// TIA Portal V20 export
ORGANIZATION_BLOCK "Startup"   // OB1060, LAD, Startup
TITLE = "Complete Restart"
AUTHOR : ERsystem_FA2_DH. Kim
// stored: AutoNumber false, IsIECCheckEnabled true, Namespace Unit1.Em6, SetENOAutomatically false
   VAR_INPUT
      LostRetentive : Bool;   // True if retentive data are lost
      LostRTC : Bool;   // True if date and time are lost
   END_VAR
BEGIN

REGION Network 1 (SCL): Build the Absolut Reference Designator
   // Set the Absoult Reference Designator in the Config DB
   IF LEN(IN := "Unit1.Em6.Config".em.referenceDesignator.parent) <> 0 THEN
     "Unit1.Em6.Config".em.referenceDesignator.combined := CONCAT_WSTRING(IN1 := "Unit1.Em6.Config".em.referenceDesignator.parent, IN2 := WSTRING#'.', IN3 := "Unit1.Em6.Config".em.referenceDesignator.relative);
   ELSE
     "Unit1.Em6.Config".em.referenceDesignator.combined := "Unit1.Em6.Config".em.referenceDesignator.relative;
   END_IF;
END_REGION

REGION Network 2 (SCL): Assign axes data
   //Assign axes
   "Unit1.Em6.Config".axis[1] := "BA030AZSCDR21_FinalRollerFrontAxisX";
   "Unit1.Em6.Config".axis[2] := "BA030AZSCDR22_FinalRollerRearAxisX";
   "Unit1.Em6.Config".axis[3] := "BA030AZSCDR23_MendrelAnodeFrontAxisY";
   "Unit1.Em6.Config".axis[4] := "BA030AZSCDR24_MendrelAnodeFrontAxisZ";
   "Unit1.Em6.Config".axis[5] := "BA030AZSCDR25_MendrelAnodeRearAxisY";
   "Unit1.Em6.Config".axis[6] := "BA030AZSCDR26_MendrelAnodeRearAxisZ";
   "Unit1.Em6.Config".axis[7] := "BA030AZSCDR27_MendrelCathodeFrontAxisY";
   "Unit1.Em6.Config".axis[8] := "BA030AZSCDR28_MendrelCathodeFrontAxisZ";
   "Unit1.Em6.Config".axis[9] := "BA030AZSCDR29_MendrelCathodeRearAxisY";
   "Unit1.Em6.Config".axis[10] := "BA030AZSCDR30_MendrelCathodeRearAxisZ";
   "Unit1.Em6.Config".axis[11] := "BA030AZSCDR31_StackTableAxisZ";
   "Unit1.Em6.Config".axis[12] := "BA030AZSCDR32_StackTableOutFrontAxisZ";
   "Unit1.Em6.Config".axis[13] := "BA030AZSCDR33_StackTableOutRearAxisZ";
   "Unit1.Em6.Config".axis[14] := "BA030A_MasterAxis";

   // Config.cam[1] := _.BA030AZSCDR21_FinalRollerFrontXCamMain;
   // Config.cam[2] := _.BA030AZSCDR23_MendrelAnodeFrontAxisYCamMain;
   // Config.cam[3] := _.BA030AZSCDR24_MendrelAnodeFrontAxisZCamMain;
   // Config.cam[4] := _.BA030AZSCDR25_MendrelAnodeRearAxisYCamMain;
   // Config.cam[5] := _.BA030AZSCDR26_MendrelAnodeRearAxisZCamMain;
   // Config.cam[6] := _.BA030AZSCDR23_MendrelCathodeFrontAxisYCamMain;
   // Config.cam[7] := _.BA030AZSCDR24_MendrelCathodeFrontAxisZCamMain;
   // Config.cam[8] := _.BA030AZSCDR25_MendrelCathodeRearAxisYCamMain;
   // Config.cam[9] := _.BA030AZSCDR26_MendrelCathodeRearAxisZCamMain;

   // FB Enable
   "Unit1.Em6.HmiInterface".cmFinalRollerFrontAxisX.commands.enableMasterControl := TRUE;
   "Unit1.Em6.HmiInterface".cmFinalRollerRearAxisX.commands.enableMasterControl := TRUE;
   "Unit1.Em6.HmiInterface".cmMendrelAnodeFrontAxisY.commands.enableMasterControl := TRUE;
   "Unit1.Em6.HmiInterface".cmMendrelAnodeFrontAxisZ.commands.enableMasterControl := TRUE;
   "Unit1.Em6.HmiInterface".cmMendrelAnodeRearAxisY.commands.enableMasterControl := TRUE;
   "Unit1.Em6.HmiInterface".cmMendrelAnodeRearAxisZ.commands.enableMasterControl := TRUE;
   "Unit1.Em6.HmiInterface".cmMendrelCathodeFrontAxisY.commands.enableMasterControl := TRUE;
   "Unit1.Em6.HmiInterface".cmMendrelCathodeFrontAxisZ.commands.enableMasterControl := TRUE;
   "Unit1.Em6.HmiInterface".cmMendrelCathodeRearAxisY.commands.enableMasterControl := TRUE;
   "Unit1.Em6.HmiInterface".cmMendrelCathodeRearAxisZ.commands.enableMasterControl := TRUE;
   "Unit1.Em6.HmiInterface".cmStackTableAxisZ.commands.enableMasterControl := TRUE;
   "Unit1.Em6.HmiInterface".cmStackTableOutFrontAxisZ.commands.enableMasterControl := TRUE;
   "Unit1.Em6.HmiInterface".cmStackTableOutRearAxisZ.commands.enableMasterControl := TRUE;

   // Axis 1 BA040AZSCDR21_FinalRollerFrontAxisX
   "Unit1.Em6.HmiInterface".cmFinalRollerFrontAxisX.commandConfiguration.jog.velocity := 10.0;
   "Unit1.Em6.HmiInterface".cmFinalRollerFrontAxisX.commandConfiguration.jog.acceleration := 100.0;
   "Unit1.Em6.HmiInterface".cmFinalRollerFrontAxisX.commandConfiguration.jog.deceleration := 100.0;
   "Unit1.Em6.HmiInterface".cmFinalRollerFrontAxisX.commandConfiguration.moveVelocity.velocity := 10.0;
   "Unit1.Em6.HmiInterface".cmFinalRollerFrontAxisX.commandConfiguration.moveVelocity.acceleration := 100.0;
   "Unit1.Em6.HmiInterface".cmFinalRollerFrontAxisX.commandConfiguration.moveVelocity.deceleration := 100.0;
   "Unit1.Em6.HmiInterface".cmFinalRollerFrontAxisX.commandConfiguration.posRelative.velocity := 10.0;
   "Unit1.Em6.HmiInterface".cmFinalRollerFrontAxisX.commandConfiguration.posRelative.acceleration := 100.0;
   "Unit1.Em6.HmiInterface".cmFinalRollerFrontAxisX.commandConfiguration.posRelative.deceleration := 100.0;
   "Unit1.Em6.HmiInterface".cmFinalRollerFrontAxisX.configuration.setPositions[0].name := 'cathode';
   "Unit1.Em6.HmiInterface".cmFinalRollerFrontAxisX.configuration.setPositions[1].name := 'anode';

   // Axis 2 BA040AZSCDR22_FinalRollerRearAxisX
   "Unit1.Em6.HmiInterface".cmFinalRollerRearAxisX.commandConfiguration.jog.velocity := 10.0;
   "Unit1.Em6.HmiInterface".cmFinalRollerRearAxisX.commandConfiguration.jog.acceleration := 100.0;
   "Unit1.Em6.HmiInterface".cmFinalRollerRearAxisX.commandConfiguration.jog.deceleration := 100.0;
   "Unit1.Em6.HmiInterface".cmFinalRollerRearAxisX.commandConfiguration.moveVelocity.velocity := 10.0;
   "Unit1.Em6.HmiInterface".cmFinalRollerRearAxisX.commandConfiguration.moveVelocity.acceleration := 100.0;
   "Unit1.Em6.HmiInterface".cmFinalRollerRearAxisX.commandConfiguration.moveVelocity.deceleration := 100.0;
   "Unit1.Em6.HmiInterface".cmFinalRollerRearAxisX.commandConfiguration.posRelative.velocity := 10.0;
   "Unit1.Em6.HmiInterface".cmFinalRollerRearAxisX.commandConfiguration.posRelative.acceleration := 100.0;
   "Unit1.Em6.HmiInterface".cmFinalRollerRearAxisX.commandConfiguration.posRelative.deceleration := 100.0;
   "Unit1.Em6.HmiInterface".cmFinalRollerRearAxisX.configuration.setPositions[0].name := 'cathode';
   "Unit1.Em6.HmiInterface".cmFinalRollerRearAxisX.configuration.setPositions[1].name := 'anode';

   // Axis 3 BA040AZSCDR23_MendrelAnodeFrontAxisY
   "Unit1.Em6.HmiInterface".cmMendrelAnodeFrontAxisY.commandConfiguration.jog.velocity := 10.0;
   "Unit1.Em6.HmiInterface".cmMendrelAnodeFrontAxisY.commandConfiguration.jog.acceleration := 100.0;
   "Unit1.Em6.HmiInterface".cmMendrelAnodeFrontAxisY.commandConfiguration.jog.deceleration := 100.0;
   "Unit1.Em6.HmiInterface".cmMendrelAnodeFrontAxisY.commandConfiguration.moveVelocity.velocity := 10.0;
   "Unit1.Em6.HmiInterface".cmMendrelAnodeFrontAxisY.commandConfiguration.moveVelocity.acceleration := 100.0;
   "Unit1.Em6.HmiInterface".cmMendrelAnodeFrontAxisY.commandConfiguration.moveVelocity.deceleration := 100.0;
   "Unit1.Em6.HmiInterface".cmMendrelAnodeFrontAxisY.commandConfiguration.posRelative.velocity := 10.0;
   "Unit1.Em6.HmiInterface".cmMendrelAnodeFrontAxisY.commandConfiguration.posRelative.acceleration := 100.0;
   "Unit1.Em6.HmiInterface".cmMendrelAnodeFrontAxisY.commandConfiguration.posRelative.deceleration := 100.0;
   "Unit1.Em6.HmiInterface".cmMendrelAnodeFrontAxisY.configuration.setPositions[0].name := 'backward';
   "Unit1.Em6.HmiInterface".cmMendrelAnodeFrontAxisY.configuration.setPositions[1].name := 'forward';

   // Axis 4 BA040AZSCDR24_MendrelAnodeFrontAxisZ
   "Unit1.Em6.HmiInterface".cmMendrelAnodeFrontAxisZ.commandConfiguration.jog.velocity := 10.0;
   "Unit1.Em6.HmiInterface".cmMendrelAnodeFrontAxisZ.commandConfiguration.jog.acceleration := 100.0;
   "Unit1.Em6.HmiInterface".cmMendrelAnodeFrontAxisZ.commandConfiguration.jog.deceleration := 100.0;
   "Unit1.Em6.HmiInterface".cmMendrelAnodeFrontAxisZ.commandConfiguration.moveVelocity.velocity := 10.0;
   "Unit1.Em6.HmiInterface".cmMendrelAnodeFrontAxisZ.commandConfiguration.moveVelocity.acceleration := 100.0;
   "Unit1.Em6.HmiInterface".cmMendrelAnodeFrontAxisZ.commandConfiguration.moveVelocity.deceleration := 100.0;
   "Unit1.Em6.HmiInterface".cmMendrelAnodeFrontAxisZ.commandConfiguration.posRelative.velocity := 10.0;
   "Unit1.Em6.HmiInterface".cmMendrelAnodeFrontAxisZ.commandConfiguration.posRelative.acceleration := 100.0;
   "Unit1.Em6.HmiInterface".cmMendrelAnodeFrontAxisZ.commandConfiguration.posRelative.deceleration := 100.0;
   "Unit1.Em6.HmiInterface".cmMendrelAnodeFrontAxisZ.configuration.setPositions[0].name := 'up';
   "Unit1.Em6.HmiInterface".cmMendrelAnodeFrontAxisZ.configuration.setPositions[1].name := 'down';

   // Axis 5 BA040AZSCDR25_MendrelAnodeRearAxisY
   "Unit1.Em6.HmiInterface".cmMendrelAnodeRearAxisY.commandConfiguration.jog.velocity := 10.0;
   "Unit1.Em6.HmiInterface".cmMendrelAnodeRearAxisY.commandConfiguration.jog.acceleration := 100.0;
   "Unit1.Em6.HmiInterface".cmMendrelAnodeRearAxisY.commandConfiguration.jog.deceleration := 100.0;
   "Unit1.Em6.HmiInterface".cmMendrelAnodeRearAxisY.commandConfiguration.moveVelocity.velocity := 10.0;
   "Unit1.Em6.HmiInterface".cmMendrelAnodeRearAxisY.commandConfiguration.moveVelocity.acceleration := 100.0;
   "Unit1.Em6.HmiInterface".cmMendrelAnodeRearAxisY.commandConfiguration.moveVelocity.deceleration := 100.0;
   "Unit1.Em6.HmiInterface".cmMendrelAnodeRearAxisY.commandConfiguration.posRelative.velocity := 10.0;
   "Unit1.Em6.HmiInterface".cmMendrelAnodeRearAxisY.commandConfiguration.posRelative.acceleration := 100.0;
   "Unit1.Em6.HmiInterface".cmMendrelAnodeRearAxisY.commandConfiguration.posRelative.deceleration := 100.0;
   "Unit1.Em6.HmiInterface".cmMendrelAnodeRearAxisY.configuration.setPositions[0].name := 'backward';
   "Unit1.Em6.HmiInterface".cmMendrelAnodeRearAxisY.configuration.setPositions[1].name := 'forward';

   // Axis 6 BA040AZSCDR26_MendrelAnodeRearAxisZ
   "Unit1.Em6.HmiInterface".cmMendrelAnodeRearAxisZ.commandConfiguration.jog.velocity := 10.0;
   "Unit1.Em6.HmiInterface".cmMendrelAnodeRearAxisZ.commandConfiguration.jog.acceleration := 100.0;
   "Unit1.Em6.HmiInterface".cmMendrelAnodeRearAxisZ.commandConfiguration.jog.deceleration := 100.0;
   "Unit1.Em6.HmiInterface".cmMendrelAnodeRearAxisZ.commandConfiguration.moveVelocity.velocity := 10.0;
   "Unit1.Em6.HmiInterface".cmMendrelAnodeRearAxisZ.commandConfiguration.moveVelocity.acceleration := 100.0;
   "Unit1.Em6.HmiInterface".cmMendrelAnodeRearAxisZ.commandConfiguration.moveVelocity.deceleration := 100.0;
   "Unit1.Em6.HmiInterface".cmMendrelAnodeRearAxisZ.commandConfiguration.posRelative.velocity := 10.0;
   "Unit1.Em6.HmiInterface".cmMendrelAnodeRearAxisZ.commandConfiguration.posRelative.acceleration := 100.0;
   "Unit1.Em6.HmiInterface".cmMendrelAnodeRearAxisZ.commandConfiguration.posRelative.deceleration := 100.0;
   "Unit1.Em6.HmiInterface".cmMendrelAnodeRearAxisZ.configuration.setPositions[0].name := 'up';
   "Unit1.Em6.HmiInterface".cmMendrelAnodeRearAxisZ.configuration.setPositions[1].name := 'down';

   // Axis 7 BA040AZSCDR27_MendrelCathodeFrontAxisY
   "Unit1.Em6.HmiInterface".cmMendrelCathodeFrontAxisY.commandConfiguration.jog.velocity := 10.0;
   "Unit1.Em6.HmiInterface".cmMendrelCathodeFrontAxisY.commandConfiguration.jog.acceleration := 100.0;
   "Unit1.Em6.HmiInterface".cmMendrelCathodeFrontAxisY.commandConfiguration.jog.deceleration := 100.0;
   "Unit1.Em6.HmiInterface".cmMendrelCathodeFrontAxisY.commandConfiguration.moveVelocity.velocity := 10.0;
   "Unit1.Em6.HmiInterface".cmMendrelCathodeFrontAxisY.commandConfiguration.moveVelocity.acceleration := 100.0;
   "Unit1.Em6.HmiInterface".cmMendrelCathodeFrontAxisY.commandConfiguration.moveVelocity.deceleration := 100.0;
   "Unit1.Em6.HmiInterface".cmMendrelCathodeFrontAxisY.commandConfiguration.posRelative.velocity := 10.0;
   "Unit1.Em6.HmiInterface".cmMendrelCathodeFrontAxisY.commandConfiguration.posRelative.acceleration := 100.0;
   "Unit1.Em6.HmiInterface".cmMendrelCathodeFrontAxisY.commandConfiguration.posRelative.deceleration := 100.0;
   "Unit1.Em6.HmiInterface".cmMendrelCathodeFrontAxisY.configuration.setPositions[0].name := 'backward';
   "Unit1.Em6.HmiInterface".cmMendrelCathodeFrontAxisY.configuration.setPositions[1].name := 'forward';

   // Axis 8 BA040AZSCDR28_MendrelCathodeFrontAxisZ
   "Unit1.Em6.HmiInterface".cmMendrelCathodeFrontAxisZ.commandConfiguration.jog.velocity := 10.0;
   "Unit1.Em6.HmiInterface".cmMendrelCathodeFrontAxisZ.commandConfiguration.jog.acceleration := 100.0;
   "Unit1.Em6.HmiInterface".cmMendrelCathodeFrontAxisZ.commandConfiguration.jog.deceleration := 100.0;
   "Unit1.Em6.HmiInterface".cmMendrelCathodeFrontAxisZ.commandConfiguration.moveVelocity.velocity := 10.0;
   "Unit1.Em6.HmiInterface".cmMendrelCathodeFrontAxisZ.commandConfiguration.moveVelocity.acceleration := 100.0;
   "Unit1.Em6.HmiInterface".cmMendrelCathodeFrontAxisZ.commandConfiguration.moveVelocity.deceleration := 100.0;
   "Unit1.Em6.HmiInterface".cmMendrelCathodeFrontAxisZ.commandConfiguration.posRelative.velocity := 10.0;
   "Unit1.Em6.HmiInterface".cmMendrelCathodeFrontAxisZ.commandConfiguration.posRelative.acceleration := 100.0;
   "Unit1.Em6.HmiInterface".cmMendrelCathodeFrontAxisZ.commandConfiguration.posRelative.deceleration := 100.0;
   "Unit1.Em6.HmiInterface".cmMendrelCathodeFrontAxisZ.configuration.setPositions[0].name := 'up';
   "Unit1.Em6.HmiInterface".cmMendrelCathodeFrontAxisZ.configuration.setPositions[1].name := 'down';

   // Axis 9 BA040AZSCDR29_MendrelCathodeRearAxisY
   "Unit1.Em6.HmiInterface".cmMendrelCathodeRearAxisY.commandConfiguration.jog.velocity := 10.0;
   "Unit1.Em6.HmiInterface".cmMendrelCathodeRearAxisY.commandConfiguration.jog.acceleration := 100.0;
   "Unit1.Em6.HmiInterface".cmMendrelCathodeRearAxisY.commandConfiguration.jog.deceleration := 100.0;
   "Unit1.Em6.HmiInterface".cmMendrelCathodeRearAxisY.commandConfiguration.moveVelocity.velocity := 10.0;
   "Unit1.Em6.HmiInterface".cmMendrelCathodeRearAxisY.commandConfiguration.moveVelocity.acceleration := 100.0;
   "Unit1.Em6.HmiInterface".cmMendrelCathodeRearAxisY.commandConfiguration.moveVelocity.deceleration := 100.0;
   "Unit1.Em6.HmiInterface".cmMendrelCathodeRearAxisY.commandConfiguration.posRelative.velocity := 10.0;
   "Unit1.Em6.HmiInterface".cmMendrelCathodeRearAxisY.commandConfiguration.posRelative.acceleration := 100.0;
   "Unit1.Em6.HmiInterface".cmMendrelCathodeRearAxisY.commandConfiguration.posRelative.deceleration := 100.0;
   "Unit1.Em6.HmiInterface".cmMendrelCathodeRearAxisY.configuration.setPositions[0].name := 'backward';
   "Unit1.Em6.HmiInterface".cmMendrelCathodeRearAxisY.configuration.setPositions[1].name := 'forward';

   // Axis 10 BA040AZSCDR30_MendrelCathodeRearAxisZ
   "Unit1.Em6.HmiInterface".cmMendrelCathodeRearAxisZ.commandConfiguration.jog.velocity := 10.0;
   "Unit1.Em6.HmiInterface".cmMendrelCathodeRearAxisZ.commandConfiguration.jog.acceleration := 100.0;
   "Unit1.Em6.HmiInterface".cmMendrelCathodeRearAxisZ.commandConfiguration.jog.deceleration := 100.0;
   "Unit1.Em6.HmiInterface".cmMendrelCathodeRearAxisZ.commandConfiguration.moveVelocity.velocity := 10.0;
   "Unit1.Em6.HmiInterface".cmMendrelCathodeRearAxisZ.commandConfiguration.moveVelocity.acceleration := 100.0;
   "Unit1.Em6.HmiInterface".cmMendrelCathodeRearAxisZ.commandConfiguration.moveVelocity.deceleration := 100.0;
   "Unit1.Em6.HmiInterface".cmMendrelCathodeRearAxisZ.commandConfiguration.posRelative.velocity := 10.0;
   "Unit1.Em6.HmiInterface".cmMendrelCathodeRearAxisZ.commandConfiguration.posRelative.acceleration := 100.0;
   "Unit1.Em6.HmiInterface".cmMendrelCathodeRearAxisZ.commandConfiguration.posRelative.deceleration := 100.0;
   "Unit1.Em6.HmiInterface".cmMendrelCathodeRearAxisZ.configuration.setPositions[0].name := 'up';
   "Unit1.Em6.HmiInterface".cmMendrelCathodeRearAxisZ.configuration.setPositions[1].name := 'down';

   // Axis 11 BA040AZSCDR31_StackTableAxisZ
   "Unit1.Em6.HmiInterface".cmStackTableAxisZ.commandConfiguration.jog.velocity := 10.0;
   "Unit1.Em6.HmiInterface".cmStackTableAxisZ.commandConfiguration.jog.acceleration := 100.0;
   "Unit1.Em6.HmiInterface".cmStackTableAxisZ.commandConfiguration.jog.deceleration := 100.0;
   "Unit1.Em6.HmiInterface".cmStackTableAxisZ.commandConfiguration.moveVelocity.velocity := 10.0;
   "Unit1.Em6.HmiInterface".cmStackTableAxisZ.commandConfiguration.moveVelocity.acceleration := 100.0;
   "Unit1.Em6.HmiInterface".cmStackTableAxisZ.commandConfiguration.moveVelocity.deceleration := 100.0;
   "Unit1.Em6.HmiInterface".cmStackTableAxisZ.commandConfiguration.posRelative.velocity := 10.0;
   "Unit1.Em6.HmiInterface".cmStackTableAxisZ.commandConfiguration.posRelative.acceleration := 100.0;
   "Unit1.Em6.HmiInterface".cmStackTableAxisZ.commandConfiguration.posRelative.deceleration := 100.0;
   "Unit1.Em6.HmiInterface".cmStackTableAxisZ.configuration.setPositions[0].name := 'wait';
   "Unit1.Em6.HmiInterface".cmStackTableAxisZ.configuration.setPositions[1].name := 'currentJRThickness';
   "Unit1.Em6.HmiInterface".cmStackTableAxisZ.configuration.setPositions[2].name := 'fullJRThickness';

   // Axis 12 BA040AZSCDR32_StackTableOutFrontAxisZ
   "Unit1.Em6.HmiInterface".cmStackTableOutFrontAxisZ.commandConfiguration.jog.velocity := 10.0;
   "Unit1.Em6.HmiInterface".cmStackTableOutFrontAxisZ.commandConfiguration.jog.acceleration := 100.0;
   "Unit1.Em6.HmiInterface".cmStackTableOutFrontAxisZ.commandConfiguration.jog.deceleration := 100.0;
   "Unit1.Em6.HmiInterface".cmStackTableOutFrontAxisZ.commandConfiguration.moveVelocity.velocity := 10.0;
   "Unit1.Em6.HmiInterface".cmStackTableOutFrontAxisZ.commandConfiguration.moveVelocity.acceleration := 100.0;
   "Unit1.Em6.HmiInterface".cmStackTableOutFrontAxisZ.commandConfiguration.moveVelocity.deceleration := 100.0;
   "Unit1.Em6.HmiInterface".cmStackTableOutFrontAxisZ.commandConfiguration.posRelative.velocity := 10.0;
   "Unit1.Em6.HmiInterface".cmStackTableOutFrontAxisZ.commandConfiguration.posRelative.acceleration := 100.0;
   "Unit1.Em6.HmiInterface".cmStackTableOutFrontAxisZ.commandConfiguration.posRelative.deceleration := 100.0;
   "Unit1.Em6.HmiInterface".cmStackTableOutFrontAxisZ.configuration.setPositions[0].name := 'down';
   "Unit1.Em6.HmiInterface".cmStackTableOutFrontAxisZ.configuration.setPositions[1].name := 'up';

   // Axis 13 BA040AZSCDR33_StackTableOutRearAxisZ
   "Unit1.Em6.HmiInterface".cmStackTableOutRearAxisZ.commandConfiguration.jog.velocity := 10.0;
   "Unit1.Em6.HmiInterface".cmStackTableOutRearAxisZ.commandConfiguration.jog.acceleration := 100.0;
   "Unit1.Em6.HmiInterface".cmStackTableOutRearAxisZ.commandConfiguration.jog.deceleration := 100.0;
   "Unit1.Em6.HmiInterface".cmStackTableOutRearAxisZ.commandConfiguration.moveVelocity.velocity := 10.0;
   "Unit1.Em6.HmiInterface".cmStackTableOutRearAxisZ.commandConfiguration.moveVelocity.acceleration := 100.0;
   "Unit1.Em6.HmiInterface".cmStackTableOutRearAxisZ.commandConfiguration.moveVelocity.deceleration := 100.0;
   "Unit1.Em6.HmiInterface".cmStackTableOutRearAxisZ.commandConfiguration.posRelative.velocity := 10.0;
   "Unit1.Em6.HmiInterface".cmStackTableOutRearAxisZ.commandConfiguration.posRelative.acceleration := 100.0;
   "Unit1.Em6.HmiInterface".cmStackTableOutRearAxisZ.commandConfiguration.posRelative.deceleration := 100.0;
   "Unit1.Em6.HmiInterface".cmStackTableOutRearAxisZ.configuration.setPositions[0].name := 'down';
   "Unit1.Em6.HmiInterface".cmStackTableOutRearAxisZ.configuration.setPositions[1].name := 'up';
END_REGION

REGION Network 3 (SCL): Assign TwoWayActuator data
   //Assign Configuration data of TwoWayActuator

   //cmMendrelAnodeFrontClamp
   "Unit1.Em6.Config".cmMendrelAnodeFrontClamp.referenceDesignator := WSTRING#'AnodeFrontClamp';
   "Unit1.Em6.Config".cmMendrelAnodeFrontClamp.disableFeedbackHomePos := TRUE;
   "Unit1.Em6.Config".cmMendrelAnodeFrontClamp.disableFeedbackWorkPos := TRUE;
   "Unit1.Em6.HmiInterface".cmMendrelAnodeFrontClamp.configuration.referenceDesignator := WSTRING#'AnodeFrontClamp';
   "Unit1.Em6.HmiInterface".cmMendrelAnodeFrontClamp.configuration.disableFeedbackHomePos := TRUE;
   "Unit1.Em6.HmiInterface".cmMendrelAnodeFrontClamp.configuration.disableFeedbackWorkPos := TRUE;

   //cmMendrelAnodeRearClamp
   "Unit1.Em6.Config".cmMendrelAnodeRearClamp.referenceDesignator := WSTRING#'AnodeRearClamp';
   "Unit1.Em6.Config".cmMendrelAnodeRearClamp.disableFeedbackHomePos := TRUE;
   "Unit1.Em6.Config".cmMendrelAnodeRearClamp.disableFeedbackWorkPos := TRUE;
   "Unit1.Em6.HmiInterface".cmMendrelAnodeRearClamp.configuration.referenceDesignator := WSTRING#'AnodeRearClamp';
   "Unit1.Em6.HmiInterface".cmMendrelAnodeRearClamp.configuration.disableFeedbackHomePos := TRUE;
   "Unit1.Em6.HmiInterface".cmMendrelAnodeRearClamp.configuration.disableFeedbackWorkPos := TRUE;

   //cmMendrelCathodeFrontClamp
   "Unit1.Em6.Config".cmMendrelCathodeFrontClamp.referenceDesignator := WSTRING#'CathodeFrontClamp';
   "Unit1.Em6.Config".cmMendrelCathodeFrontClamp.disableFeedbackHomePos := TRUE;
   "Unit1.Em6.Config".cmMendrelCathodeFrontClamp.disableFeedbackWorkPos := TRUE;
   "Unit1.Em6.HmiInterface".cmMendrelCathodeFrontClamp.configuration.referenceDesignator := WSTRING#'CathodeFrontClamp';
   "Unit1.Em6.HmiInterface".cmMendrelCathodeFrontClamp.configuration.disableFeedbackHomePos := TRUE;
   "Unit1.Em6.HmiInterface".cmMendrelCathodeFrontClamp.configuration.disableFeedbackWorkPos := TRUE;

   //cmMendrelCathodeRearClamp
   "Unit1.Em6.Config".cmMendrelCathodeRearClamp.referenceDesignator := WSTRING#'CathodeRearClamp';
   "Unit1.Em6.Config".cmMendrelCathodeRearClamp.disableFeedbackHomePos := TRUE;
   "Unit1.Em6.Config".cmMendrelCathodeRearClamp.disableFeedbackWorkPos := TRUE;
   "Unit1.Em6.HmiInterface".cmMendrelCathodeRearClamp.configuration.referenceDesignator := WSTRING#'CathodeRearClamp';
   "Unit1.Em6.HmiInterface".cmMendrelCathodeRearClamp.configuration.disableFeedbackHomePos := TRUE;
   "Unit1.Em6.HmiInterface".cmMendrelCathodeRearClamp.configuration.disableFeedbackWorkPos := TRUE;

   //cmStackTableVaccum
   "Unit1.Em6.Config".cmStackTableVaccum.referenceDesignator := WSTRING#'StackTableVaccum';
   "Unit1.Em6.Config".cmStackTableVaccum.disableFeedbackHomePos := FALSE;
   "Unit1.Em6.Config".cmStackTableVaccum.disableFeedbackWorkPos := FALSE;
   "Unit1.Em6.HmiInterface".cmStackTableVaccum.configuration.referenceDesignator := WSTRING#'StackTableVaccum';
   "Unit1.Em6.HmiInterface".cmStackTableVaccum.configuration.disableFeedbackHomePos := FALSE;
   "Unit1.Em6.HmiInterface".cmStackTableVaccum.configuration.disableFeedbackWorkPos := FALSE;

   //cmStackTableGapPadUpDown
   "Unit1.Em6.Config".cmStackTableGapPadUpDown.referenceDesignator := WSTRING#'GapPadUpDown';
   "Unit1.Em6.Config".cmStackTableGapPadUpDown.disableFeedbackHomePos := FALSE;
   "Unit1.Em6.Config".cmStackTableGapPadUpDown.disableFeedbackWorkPos := FALSE;
   "Unit1.Em6.HmiInterface".cmStackTableGapPadUpDown.configuration.referenceDesignator := WSTRING#'GapPadUpDown';
   "Unit1.Em6.HmiInterface".cmStackTableGapPadUpDown.configuration.disableFeedbackHomePos := FALSE;
   "Unit1.Em6.HmiInterface".cmStackTableGapPadUpDown.configuration.disableFeedbackWorkPos := FALSE;
END_REGION
END_ORGANIZATION_BLOCK
